FUNCTION_BLOCK ABSTRACT FB_Car
VAR_INPUT
END_VAR
VAR_OUTPUT
END_VAR
VAR
END_VAR

METHOD Running : BOOL
VAR_INPUT
END_VAR
END_METHOD

METHOD ABSTRACT Start : BOOL
VAR_INPUT
END_VAR
END_METHOD

END_FUNCTION_BLOCK

(* stored: Version 1.1.0.1, ProductVersion 3.1.4024.16
   POU FB_Car: Id {7204386d-eef9-428d-9a12-9c863ebad0ab}, SpecialFunc None
   Method Running: Id {a9c4540a-b3c4-4ff9-a5b7-95c3ea3c4cf5}
   Method Start: Id {a27c00aa-7d49-4168-a041-860d21db2d4c} *)
